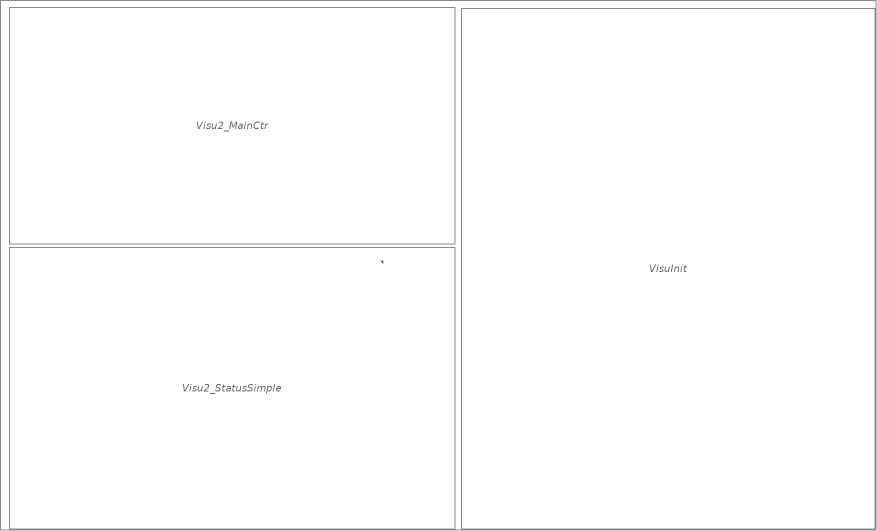
VISUALIZATION Visualization  // 877x531
    Button (382,261 1x2)
    TabControl (9,7 446x237)
        shows Visu2_MainCtr()
        shows Visu2_LanguageUser()
        [0]: TabTitle=MainControl
        [1]: TabTitle=Language / User
    TabControl (461,8 414x521), frame switch variable: stParam.stStatus.eMMA
        shows VisuInit()
        shows VisuAuto()
        shows VisuManual()
        [0]: TabTitle=Init
        [1]: TabTitle=Auto
        [2]: TabTitle=Manual
    TabControl (9,247 446x282)
        shows Visu2_StatusSimple()
        shows Visu2_Status()
        [0]: TabTitle=Status Simple
        [1]: TabTitle=Status Full
END_VISUALIZATION

(* stored: Version 1.1.0.1, ProductVersion 3.1.4020.12
   Visu Visualization: Id {1e4c2f99-d035-41f9-adba-3d4322eca24e} *)
